      - frame TeachingPoints_16-06-04 at (12133.67, 1957.34, 973.56) mm, rotated rx 180 ry 0 rz 0 deg
        - target Point_16-06-04 (Cartesian target) at (0, 0, 0) mm; joints [12200, 3550, 510] of gantry
      - frame TeachingPoints_17-06-04 at (12633.67, 1957.34, 973.56) mm, rotated rx 180 ry 0 rz 0 deg
        - target Point_17-06-04 (Cartesian target) at (0, 0, 0) mm; joints [12700, 3550, 510] of gantry
      - frame TeachingPoints_18-06-04 at (13133.67, 1957.34, 973.56) mm, rotated rx 180 ry 0 rz 0 deg
        - target Point_18-06-04 (Cartesian target) at (0, 0, 0) mm; joints [13200, 3550, 510] of gantry
      - frame TeachingPoints_19-06-04 at (13633.67, 1957.34, 973.56) mm, rotated rx 180 ry 0 rz 0 deg
        - target Point_19-06-04 (Cartesian target) at (0, 0, 0) mm; joints [13700, 3550, 510] of gantry
      - frame TeachingPoints_20-06-04 at (14133.67, 1957.34, 973.56) mm, rotated rx 180 ry 0 rz 0 deg
        - target Point_20-06-04 (Cartesian target) at (0, 0, 0) mm; joints [14200, 3550, 510] of gantry
      - frame TeachingPoints_01-01-05 at (4633.67, 4457.34, 1108.56) mm, rotated rx 180 ry 0 rz 0 deg
        - target Point_01-01-05 (Cartesian target) at (0, 0, 0) mm; joints [4700, 1050, 375] of gantry
      - frame TeachingPoints_02-01-05 at (5133.67, 4457.34, 1108.56) mm, rotated rx 180 ry 0 rz 0 deg
        - target Point_02-01-05 (Cartesian target) at (0, 0, 0) mm; joints [5200, 1050, 375] of gantry
      - frame TeachingPoints_03-01-05 at (5633.67, 4457.34, 1108.56) mm, rotated rx 180 ry 0 rz 0 deg
        - target Point_03-01-05 (Cartesian target) at (0, 0, 0) mm; joints [5700, 1050, 375] of gantry
      - frame TeachingPoints_04-01-05 at (6133.67, 4457.34, 1108.56) mm, rotated rx 180 ry 0 rz 0 deg
        - target Point_04-01-05 (Cartesian target) at (0, 0, 0) mm; joints [6200, 1050, 375] of gantry
      - frame TeachingPoints_05-01-05 at (6633.67, 4457.34, 1108.56) mm, rotated rx 180 ry 0 rz 0 deg
        - target Point_05-01-05 (Cartesian target) at (0, 0, 0) mm; joints [6700, 1050, 375] of gantry
      - frame TeachingPoints_06-01-05 at (7133.67, 4457.34, 1108.56) mm, rotated rx 180 ry 0 rz 0 deg
        - target Point_06-01-05 (Cartesian target) at (0, 0, 0) mm; joints [7200, 1050, 375] of gantry
      - frame TeachingPoints_07-01-05 at (7633.67, 4457.34, 1108.56) mm, rotated rx 180 ry 0 rz 0 deg
        - target Point_07-01-05 (Cartesian target) at (0, 0, 0) mm; joints [7700, 1050, 375] of gantry
      - frame TeachingPoints_08-01-05 at (8133.67, 4457.34, 1108.56) mm, rotated rx 180 ry 0 rz 0 deg
        - target Point_08-01-05 (Cartesian target) at (0, 0, 0) mm; joints [8200, 1050, 375] of gantry
      - frame TeachingPoints_09-01-05 at (8633.67, 4457.34, 1108.56) mm, rotated rx 180 ry 0 rz 0 deg
        - target Point_09-01-05 (Cartesian target) at (0, 0, 0) mm; joints [8700, 1050, 375] of gantry
      - frame TeachingPoints_10-01-05 at (9133.67, 4457.34, 1108.56) mm, rotated rx 180 ry 0 rz 0 deg
        - target Point_10-01-05 (Cartesian target) at (0, 0, 0) mm; joints [9200, 1050, 375] of gantry
      - frame TeachingPoints_11-01-05 at (9633.67, 4457.34, 1108.56) mm, rotated rx 180 ry 0 rz 0 deg
        - target Point_11-01-05 (Cartesian target) at (0, 0, 0) mm; joints [9700, 1050, 375] of gantry
      - frame TeachingPoints_12-01-05 at (10133.67, 4457.34, 1108.56) mm, rotated rx 180 ry 0 rz 0 deg
        - target Point_12-01-05 (Cartesian target) at (0, 0, 0) mm; joints [10200, 1050, 375] of gantry
      - frame TeachingPoints_13-01-05 at (10633.67, 4457.34, 1108.56) mm, rotated rx 180 ry 0 rz 0 deg
        - target Point_13-01-05 (Cartesian target) at (0, 0, 0) mm; joints [10700, 1050, 375] of gantry
      - frame TeachingPoints_14-01-05 at (11133.67, 4457.34, 1108.56) mm, rotated rx 180 ry 0 rz 0 deg
        - target Point_14-01-05 (Cartesian target) at (0, 0, 0) mm; joints [11200, 1050, 375] of gantry
      - frame TeachingPoints_15-01-05 at (11633.67, 4457.34, 1108.56) mm, rotated rx 180 ry 0 rz 0 deg
        - target Point_15-01-05 (Cartesian target) at (0, 0, 0) mm; joints [11700, 1050, 375] of gantry
      - frame TeachingPoints_16-01-05 at (12133.67, 4457.34, 1108.56) mm, rotated rx 180 ry 0 rz 0 deg
        - target Point_16-01-05 (Cartesian target) at (0, 0, 0) mm; joints [12200, 1050, 375] of gantry
      - frame TeachingPoints_17-01-05 at (12633.67, 4457.34, 1108.56) mm, rotated rx 180 ry 0 rz 0 deg
        - target Point_17-01-05 (Cartesian target) at (0, 0, 0) mm; joints [12700, 1050, 375] of gantry
      - frame TeachingPoints_18-01-05 at (13133.67, 4457.34, 1108.56) mm, rotated rx 180 ry 0 rz 0 deg
        - target Point_18-01-05 (Cartesian target) at (0, 0, 0) mm; joints [13200, 1050, 375] of gantry
      - frame TeachingPoints_19-01-05 at (13633.67, 4457.34, 1108.56) mm, rotated rx 180 ry 0 rz 0 deg
        - target Point_19-01-05 (Cartesian target) at (0, 0, 0) mm; joints [13700, 1050, 375] of gantry
      - frame TeachingPoints_20-01-05 at (14133.67, 4457.34, 1108.56) mm, rotated rx 180 ry 0 rz 0 deg
        - target Point_20-01-05 (Cartesian target) at (0, 0, 0) mm; joints [14200, 1050, 375] of gantry
      - frame TeachingPoints_01-02-05 at (4633.67, 3957.34, 1108.56) mm, rotated rx 180 ry 0 rz 0 deg
        - target Point_01-02-05 (Cartesian target) at (0, 0, 0) mm; joints [4700, 1550, 375] of gantry
      - frame TeachingPoints_02-02-05 at (5133.67, 3957.34, 1108.56) mm, rotated rx 180 ry 0 rz 0 deg
        - target Point_02-02-05 (Cartesian target) at (0, 0, 0) mm; joints [5200, 1550, 375] of gantry
      - frame TeachingPoints_03-02-05 at (5633.67, 3957.34, 1108.56) mm, rotated rx 180 ry 0 rz 0 deg
        - target Point_03-02-05 (Cartesian target) at (0, 0, 0) mm; joints [5700, 1550, 375] of gantry
      - frame TeachingPoints_04-02-05 at (6133.67, 3957.34, 1108.56) mm, rotated rx 180 ry 0 rz 0 deg
        - target Point_04-02-05 (Cartesian target) at (0, 0, 0) mm; joints [6200, 1550, 375] of gantry
      - frame TeachingPoints_05-02-05 at (6633.67, 3957.34, 1108.56) mm, rotated rx 180 ry 0 rz 0 deg
        - target Point_05-02-05 (Cartesian target) at (0, 0, 0) mm; joints [6700, 1550, 375] of gantry
      - frame TeachingPoints_06-02-05 at (7133.67, 3957.34, 1108.56) mm, rotated rx 180 ry 0 rz 0 deg
        - target Point_06-02-05 (Cartesian target) at (0, 0, 0) mm; joints [7200, 1550, 375] of gantry
      - frame TeachingPoints_07-02-05 at (7633.67, 3957.34, 1108.56) mm, rotated rx 180 ry 0 rz 0 deg
        - target Point_07-02-05 (Cartesian target) at (0, 0, 0) mm; joints [7700, 1550, 375] of gantry
      - frame TeachingPoints_08-02-05 at (8133.67, 3957.34, 1108.56) mm, rotated rx 180 ry 0 rz 0 deg
        - target Point_08-02-05 (Cartesian target) at (0, 0, 0) mm; joints [8200, 1550, 375] of gantry
      - frame TeachingPoints_09-02-05 at (8633.67, 3957.34, 1108.56) mm, rotated rx 180 ry 0 rz 0 deg
        - target Point_09-02-05 (Cartesian target) at (0, 0, 0) mm; joints [8700, 1550, 375] of gantry
      - frame TeachingPoints_10-02-05 at (9133.67, 3957.34, 1108.56) mm, rotated rx 180 ry 0 rz 0 deg
        - target Point_10-02-05 (Cartesian target) at (0, 0, 0) mm; joints [9200, 1550, 375] of gantry
      - frame TeachingPoints_11-02-05 at (9633.67, 3957.34, 1108.56) mm, rotated rx 180 ry 0 rz 0 deg
        - target Point_11-02-05 (Cartesian target) at (0, 0, 0) mm; joints [9700, 1550, 375] of gantry
      - frame TeachingPoints_12-02-05 at (10133.67, 3957.34, 1108.56) mm, rotated rx 180 ry 0 rz 0 deg
        - target Point_12-02-05 (Cartesian target) at (0, 0, 0) mm; joints [10200, 1550, 375] of gantry
      - frame TeachingPoints_13-02-05 at (10633.67, 3957.34, 1108.56) mm, rotated rx 180 ry 0 rz 0 deg
        - target Point_13-02-05 (Cartesian target) at (0, 0, 0) mm; joints [10700, 1550, 375] of gantry
      - frame TeachingPoints_14-02-05 at (11133.67, 3957.34, 1108.56) mm, rotated rx 180 ry 0 rz 0 deg
        - target Point_14-02-05 (Cartesian target) at (0, 0, 0) mm; joints [11200, 1550, 375] of gantry
      - frame TeachingPoints_15-02-05 at (11633.67, 3957.34, 1108.56) mm, rotated rx 180 ry 0 rz 0 deg
        - target Point_15-02-05 (Cartesian target) at (0, 0, 0) mm; joints [11700, 1550, 375] of gantry
      - frame TeachingPoints_16-02-05 at (12133.67, 3957.34, 1108.56) mm, rotated rx 180 ry 0 rz 0 deg
        - target Point_16-02-05 (Cartesian target) at (0, 0, 0) mm; joints [12200, 1550, 375] of gantry
      - frame TeachingPoints_17-02-05 at (12633.67, 3957.34, 1108.56) mm, rotated rx 180 ry 0 rz 0 deg
        - target Point_17-02-05 (Cartesian target) at (0, 0, 0) mm; joints [12700, 1550, 375] of gantry
      - frame TeachingPoints_18-02-05 at (13133.67, 3957.34, 1108.56) mm, rotated rx 180 ry 0 rz 0 deg
        - target Point_18-02-05 (Cartesian target) at (0, 0, 0) mm; joints [13200, 1550, 375] of gantry
      - frame TeachingPoints_19-02-05 at (13633.67, 3957.34, 1108.56) mm, rotated rx 180 ry 0 rz 0 deg
        - target Point_19-02-05 (Cartesian target) at (0, 0, 0) mm; joints [13700, 1550, 375] of gantry
      - frame TeachingPoints_20-02-05 at (14133.67, 3957.34, 1108.56) mm, rotated rx 180 ry 0 rz 0 deg
        - target Point_20-02-05 (Cartesian target) at (0, 0, 0) mm; joints [14200, 1550, 375] of gantry
      - frame TeachingPoints_01-03-05 at (4633.67, 3457.34, 1108.56) mm, rotated rx 180 ry 0 rz 0 deg
        - target Point_01-03-05 (Cartesian target) at (0, 0, 0) mm; joints [4700, 2050, 375] of gantry
      - frame TeachingPoints_02-03-05 at (5133.67, 3457.34, 1108.56) mm, rotated rx 180 ry 0 rz 0 deg
        - target Point_02-03-05 (Cartesian target) at (0, 0, 0) mm; joints [5200, 2050, 375] of gantry
      - frame TeachingPoints_03-03-05 at (5633.67, 3457.34, 1108.56) mm, rotated rx 180 ry 0 rz 0 deg
        - target Point_03-03-05 (Cartesian target) at (0, 0, 0) mm; joints [5700, 2050, 375] of gantry
      - frame TeachingPoints_04-03-05 at (6133.67, 3457.34, 1108.56) mm, rotated rx 180 ry 0 rz 0 deg
        - target Point_04-03-05 (Cartesian target) at (0, 0, 0) mm; joints [6200, 2050, 375] of gantry
      - frame TeachingPoints_05-03-05 at (6633.67, 3457.34, 1108.56) mm, rotated rx 180 ry 0 rz 0 deg
        - target Point_05-03-05 (Cartesian target) at (0, 0, 0) mm; joints [6700, 2050, 375] of gantry
      - frame TeachingPoints_06-03-05 at (7133.67, 3457.34, 1108.56) mm, rotated rx 180 ry 0 rz 0 deg
        - target Point_06-03-05 (Cartesian target) at (0, 0, 0) mm; joints [7200, 2050, 375] of gantry
      - frame TeachingPoints_07-03-05 at (7633.67, 3457.34, 1108.56) mm, rotated rx 180 ry 0 rz 0 deg
        - target Point_07-03-05 (Cartesian target) at (0, 0, 0) mm; joints [7700, 2050, 375] of gantry
      - frame TeachingPoints_08-03-05 at (8133.67, 3457.34, 1108.56) mm, rotated rx 180 ry 0 rz 0 deg
        - target Point_08-03-05 (Cartesian target) at (0, 0, 0) mm; joints [8200, 2050, 375] of gantry
      - frame TeachingPoints_09-03-05 at (8633.67, 3457.34, 1108.56) mm, rotated rx 180 ry 0 rz 0 deg
        - target Point_09-03-05 (Cartesian target) at (0, 0, 0) mm; joints [8700, 2050, 375] of gantry
      - frame TeachingPoints_10-03-05 at (9133.67, 3457.34, 1108.56) mm, rotated rx 180 ry 0 rz 0 deg
        - target Point_10-03-05 (Cartesian target) at (0, 0, 0) mm; joints [9200, 2050, 375] of gantry
      - frame TeachingPoints_11-03-05 at (9633.67, 3457.34, 1108.56) mm, rotated rx 180 ry 0 rz 0 deg
        - target Point_11-03-05 (Cartesian target) at (0, 0, 0) mm; joints [9700, 2050, 375] of gantry
      - frame TeachingPoints_12-03-05 at (10133.67, 3457.34, 1108.56) mm, rotated rx 180 ry 0 rz 0 deg
        - target Point_12-03-05 (Cartesian target) at (0, 0, 0) mm; joints [10200, 2050, 375] of gantry
      - frame TeachingPoints_13-03-05 at (10633.67, 3457.34, 1108.56) mm, rotated rx 180 ry 0 rz 0 deg
        - target Point_13-03-05 (Cartesian target) at (0, 0, 0) mm; joints [10700, 2050, 375] of gantry
      - frame TeachingPoints_14-03-05 at (11133.67, 3457.34, 1108.56) mm, rotated rx 180 ry 0 rz 0 deg
        - target Point_14-03-05 (Cartesian target) at (0, 0, 0) mm; joints [11200, 2050, 375] of gantry
      - frame TeachingPoints_15-03-05 at (11633.67, 3457.34, 1108.56) mm, rotated rx 180 ry 0 rz 0 deg
        - target Point_15-03-05 (Cartesian target) at (0, 0, 0) mm; joints [11700, 2050, 375] of gantry
      - frame TeachingPoints_16-03-05 at (12133.67, 3457.34, 1108.56) mm, rotated rx 180 ry 0 rz 0 deg
        - target Point_16-03-05 (Cartesian target) at (0, 0, 0) mm; joints [12200, 2050, 375] of gantry
      - frame TeachingPoints_17-03-05 at (12633.67, 3457.34, 1108.56) mm, rotated rx 180 ry 0 rz 0 deg
        - target Point_17-03-05 (Cartesian target) at (0, 0, 0) mm; joints [12700, 2050, 375] of gantry
      - frame TeachingPoints_18-03-05 at (13133.67, 3457.34, 1108.56) mm, rotated rx 180 ry 0 rz 0 deg
        - target Point_18-03-05 (Cartesian target) at (0, 0, 0) mm; joints [13200, 2050, 375] of gantry
      - frame TeachingPoints_19-03-05 at (13633.67, 3457.34, 1108.56) mm, rotated rx 180 ry 0 rz 0 deg
        - target Point_19-03-05 (Cartesian target) at (0, 0, 0) mm; joints [13700, 2050, 375] of gantry
      - frame TeachingPoints_20-03-05 at (14133.67, 3457.34, 1108.56) mm, rotated rx 180 ry 0 rz 0 deg
        - target Point_20-03-05 (Cartesian target) at (0, 0, 0) mm; joints [14200, 2050, 375] of gantry
      - frame TeachingPoints_01-04-05 at (4633.67, 2957.34, 1108.56) mm, rotated rx 180 ry 0 rz 0 deg
        - target Point_01-04-05 (Cartesian target) at (0, 0, 0) mm; joints [4700, 2550, 375] of gantry
      - frame TeachingPoints_02-04-05 at (5133.67, 2957.34, 1108.56) mm, rotated rx 180 ry 0 rz 0 deg
        - target Point_02-04-05 (Cartesian target) at (0, 0, 0) mm; joints [5200, 2550, 375] of gantry
      - frame TeachingPoints_03-04-05 at (5633.67, 2957.34, 1108.56) mm, rotated rx 180 ry 0 rz 0 deg
        - target Point_03-04-05 (Cartesian target) at (0, 0, 0) mm; joints [5700, 2550, 375] of gantry
      - frame TeachingPoints_04-04-05 at (6133.67, 2957.34, 1108.56) mm, rotated rx 180 ry 0 rz 0 deg
        - target Point_04-04-05 (Cartesian target) at (0, 0, 0) mm; joints [6200, 2550, 375] of gantry
      - frame TeachingPoints_05-04-05 at (6633.67, 2957.34, 1108.56) mm, rotated rx 180 ry 0 rz 0 deg
        - target Point_05-04-05 (Cartesian target) at (0, 0, 0) mm; joints [6700, 2550, 375] of gantry
      - frame TeachingPoints_06-04-05 at (7133.67, 2957.34, 1108.56) mm, rotated rx 180 ry 0 rz 0 deg
        - target Point_06-04-05 (Cartesian target) at (0, 0, 0) mm; joints [7200, 2550, 375] of gantry
      - frame TeachingPoints_07-04-05 at (7633.67, 2957.34, 1108.56) mm, rotated rx 180 ry 0 rz 0 deg
        - target Point_07-04-05 (Cartesian target) at (0, 0, 0) mm; joints [7700, 2550, 375] of gantry
      - frame TeachingPoints_08-04-05 at (8133.67, 2957.34, 1108.56) mm, rotated rx 180 ry 0 rz 0 deg
        - target Point_08-04-05 (Cartesian target) at (0, 0, 0) mm; joints [8200, 2550, 375] of gantry
      - frame TeachingPoints_09-04-05 at (8633.67, 2957.34, 1108.56) mm, rotated rx 180 ry 0 rz 0 deg
        - target Point_09-04-05 (Cartesian target) at (0, 0, 0) mm; joints [8700, 2550, 375] of gantry
      - frame TeachingPoints_10-04-05 at (9133.67, 2957.34, 1108.56) mm, rotated rx 180 ry 0 rz 0 deg
        - target Point_10-04-05 (Cartesian target) at (0, 0, 0) mm; joints [9200, 2550, 375] of gantry
      - frame TeachingPoints_11-04-05 at (9633.67, 2957.34, 1108.56) mm, rotated rx 180 ry 0 rz 0 deg
        - target Point_11-04-05 (Cartesian target) at (0, 0, 0) mm; joints [9700, 2550, 375] of gantry
      - frame TeachingPoints_12-04-05 at (10133.67, 2957.34, 1108.56) mm, rotated rx 180 ry 0 rz 0 deg
        - target Point_12-04-05 (Cartesian target) at (0, 0, 0) mm; joints [10200, 2550, 375] of gantry
      - frame TeachingPoints_13-04-05 at (10633.67, 2957.34, 1108.56) mm, rotated rx 180 ry 0 rz 0 deg
        - target Point_13-04-05 (Cartesian target) at (0, 0, 0) mm; joints [10700, 2550, 375] of gantry
      - frame TeachingPoints_14-04-05 at (11133.67, 2957.34, 1108.56) mm, rotated rx 180 ry 0 rz 0 deg
        - target Point_14-04-05 (Cartesian target) at (0, 0, 0) mm; joints [11200, 2550, 375] of gantry
      - frame TeachingPoints_15-04-05 at (11633.67, 2957.34, 1108.56) mm, rotated rx 180 ry 0 rz 0 deg
        - target Point_15-04-05 (Cartesian target) at (0, 0, 0) mm; joints [11700, 2550, 375] of gantry
      - frame TeachingPoints_16-04-05 at (12133.67, 2957.34, 1108.56) mm, rotated rx 180 ry 0 rz 0 deg
        - target Point_16-04-05 (Cartesian target) at (0, 0, 0) mm; joints [12200, 2550, 375] of gantry
      - frame TeachingPoints_17-04-05 at (12633.67, 2957.34, 1108.56) mm, rotated rx 180 ry 0 rz 0 deg
        - target Point_17-04-05 (Cartesian target) at (0, 0, 0) mm; joints [12700, 2550, 375] of gantry
      - frame TeachingPoints_18-04-05 at (13133.67, 2957.34, 1108.56) mm, rotated rx 180 ry 0 rz 0 deg
        - target Point_18-04-05 (Cartesian target) at (0, 0, 0) mm; joints [13200, 2550, 375] of gantry
      - frame TeachingPoints_19-04-05 at (13633.67, 2957.34, 1108.56) mm, rotated rx 180 ry 0 rz 0 deg
        - target Point_19-04-05 (Cartesian target) at (0, 0, 0) mm; joints [13700, 2550, 375] of gantry
      - frame TeachingPoints_20-04-05 at (14133.67, 2957.34, 1108.56) mm, rotated rx 180 ry 0 rz 0 deg
        - target Point_20-04-05 (Cartesian target) at (0, 0, 0) mm; joints [14200, 2550, 375] of gantry
      - frame TeachingPoints_01-05-05 at (4633.67, 2457.34, 1108.56) mm, rotated rx 180 ry 0 rz 0 deg
        - target Point_01-05-05 (Cartesian target) at (0, 0, 0) mm; joints [4700, 3050, 375] of gantry
      - frame TeachingPoints_02-05-05 at (5133.67, 2457.34, 1108.56) mm, rotated rx 180 ry 0 rz 0 deg
        - target Point_02-05-05 (Cartesian target) at (0, 0, 0) mm; joints [5200, 3050, 375] of gantry
      - frame TeachingPoints_03-05-05 at (5633.67, 2457.34, 1108.56) mm, rotated rx 180 ry 0 rz 0 deg
        - target Point_03-05-05 (Cartesian target) at (0, 0, 0) mm; joints [5700, 3050, 375] of gantry
      - frame TeachingPoints_04-05-05 at (6133.67, 2457.34, 1108.56) mm, rotated rx 180 ry 0 rz 0 deg
        - target Point_04-05-05 (Cartesian target) at (0, 0, 0) mm; joints [6200, 3050, 375] of gantry
      - frame TeachingPoints_05-05-05 at (6633.67, 2457.34, 1108.56) mm, rotated rx 180 ry 0 rz 0 deg
        - target Point_05-05-05 (Cartesian target) at (0, 0, 0) mm; joints [6700, 3050, 375] of gantry
      - frame TeachingPoints_06-05-05 at (7133.67, 2457.34, 1108.56) mm, rotated rx 180 ry 0 rz 0 deg
        - target Point_06-05-05 (Cartesian target) at (0, 0, 0) mm; joints [7200, 3050, 375] of gantry
      - frame TeachingPoints_07-05-05 at (7633.67, 2457.34, 1108.56) mm, rotated rx 180 ry 0 rz 0 deg
        - target Point_07-05-05 (Cartesian target) at (0, 0, 0) mm; joints [7700, 3050, 375] of gantry
      - frame TeachingPoints_08-05-05 at (8133.67, 2457.34, 1108.56) mm, rotated rx 180 ry 0 rz 0 deg
        - target Point_08-05-05 (Cartesian target) at (0, 0, 0) mm; joints [8200, 3050, 375] of gantry
      - frame TeachingPoints_09-05-05 at (8633.67, 2457.34, 1108.56) mm, rotated rx 180 ry 0 rz 0 deg
        - target Point_09-05-05 (Cartesian target) at (0, 0, 0) mm; joints [8700, 3050, 375] of gantry
      - frame TeachingPoints_10-05-05 at (9133.67, 2457.34, 1108.56) mm, rotated rx 180 ry 0 rz 0 deg
        - target Point_10-05-05 (Cartesian target) at (0, 0, 0) mm; joints [9200, 3050, 375] of gantry
      - frame TeachingPoints_11-05-05 at (9633.67, 2457.34, 1108.56) mm, rotated rx 180 ry 0 rz 0 deg
        - target Point_11-05-05 (Cartesian target) at (0, 0, 0) mm; joints [9700, 3050, 375] of gantry
      - frame TeachingPoints_12-05-05 at (10133.67, 2457.34, 1108.56) mm, rotated rx 180 ry 0 rz 0 deg
        - target Point_12-05-05 (Cartesian target) at (0, 0, 0) mm; joints [10200, 3050, 375] of gantry
      - frame TeachingPoints_13-05-05 at (10633.67, 2457.34, 1108.56) mm, rotated rx 180 ry 0 rz 0 deg
        - target Point_13-05-05 (Cartesian target) at (0, 0, 0) mm; joints [10700, 3050, 375] of gantry
      - frame TeachingPoints_14-05-05 at (11133.67, 2457.34, 1108.56) mm, rotated rx 180 ry 0 rz 0 deg
        - target Point_14-05-05 (Cartesian target) at (0, 0, 0) mm; joints [11200, 3050, 375] of gantry
      - frame TeachingPoints_15-05-05 at (11633.67, 2457.34, 1108.56) mm, rotated rx 180 ry 0 rz 0 deg
        - target Point_15-05-05 (Cartesian target) at (0, 0, 0) mm; joints [11700, 3050, 375] of gantry
      - frame TeachingPoints_16-05-05 at (12133.67, 2457.34, 1108.56) mm, rotated rx 180 ry 0 rz 0 deg
        - target Point_16-05-05 (Cartesian target) at (0, 0, 0) mm; joints [12200, 3050, 375] of gantry
      - frame TeachingPoints_17-05-05 at (12633.67, 2457.34, 1108.56) mm, rotated rx 180 ry 0 rz 0 deg
        - target Point_17-05-05 (Cartesian target) at (0, 0, 0) mm; joints [12700, 3050, 375] of gantry
      - frame TeachingPoints_18-05-05 at (13133.67, 2457.34, 1108.56) mm, rotated rx 180 ry 0 rz 0 deg
        - target Point_18-05-05 (Cartesian target) at (0, 0, 0) mm; joints [13200, 3050, 375] of gantry
      - frame TeachingPoints_19-05-05 at (13633.67, 2457.34, 1108.56) mm, rotated rx 180 ry 0 rz 0 deg
        - target Point_19-05-05 (Cartesian target) at (0, 0, 0) mm; joints [13700, 3050, 375] of gantry
      - frame TeachingPoints_20-05-05 at (14133.67, 2457.34, 1108.56) mm, rotated rx 180 ry 0 rz 0 deg
        - target Point_20-05-05 (Cartesian target) at (0, 0, 0) mm; joints [14200, 3050, 375] of gantry
      - frame TeachingPoints_01-06-05 at (4633.67, 1957.34, 1108.56) mm, rotated rx 180 ry 0 rz 0 deg
        - target Point_01-06-05 (Cartesian target) at (0, 0, 0) mm; joints [4700, 3550, 375] of gantry
      - frame TeachingPoints_02-06-05 at (5133.67, 1957.34, 1108.56) mm, rotated rx 180 ry 0 rz 0 deg
        - target Point_02-06-05 (Cartesian target) at (0, 0, 0) mm; joints [5200, 3550, 375] of gantry
      - frame TeachingPoints_03-06-05 at (5633.67, 1957.34, 1108.56) mm, rotated rx 180 ry 0 rz 0 deg
        - target Point_03-06-05 (Cartesian target) at (0, 0, 0) mm; joints [5700, 3550, 375] of gantry
      - frame TeachingPoints_04-06-05 at (6133.67, 1957.34, 1108.56) mm, rotated rx 180 ry 0 rz 0 deg
        - target Point_04-06-05 (Cartesian target) at (0, 0, 0) mm; joints [6200, 3550, 375] of gantry
      - frame TeachingPoints_05-06-05 at (6633.67, 1957.34, 1108.56) mm, rotated rx 180 ry 0 rz 0 deg
        - target Point_05-06-05 (Cartesian target) at (0, 0, 0) mm; joints [6700, 3550, 375] of gantry
      - frame TeachingPoints_06-06-05 at (7133.67, 1957.34, 1108.56) mm, rotated rx 180 ry 0 rz 0 deg
        - target Point_06-06-05 (Cartesian target) at (0, 0, 0) mm; joints [7200, 3550, 375] of gantry
      - frame TeachingPoints_07-06-05 at (7633.67, 1957.34, 1108.56) mm, rotated rx 180 ry 0 rz 0 deg
        - target Point_07-06-05 (Cartesian target) at (0, 0, 0) mm; joints [7700, 3550, 375] of gantry
      - frame TeachingPoints_08-06-05 at (8133.67, 1957.34, 1108.56) mm, rotated rx 180 ry 0 rz 0 deg
        - target Point_08-06-05 (Cartesian target) at (0, 0, 0) mm; joints [8200, 3550, 375] of gantry
      - frame TeachingPoints_09-06-05 at (8633.67, 1957.34, 1108.56) mm, rotated rx 180 ry 0 rz 0 deg
        - target Point_09-06-05 (Cartesian target) at (0, 0, 0) mm; joints [8700, 3550, 375] of gantry
      - frame TeachingPoints_10-06-05 at (9133.67, 1957.34, 1108.56) mm, rotated rx 180 ry 0 rz 0 deg
        - target Point_10-06-05 (Cartesian target) at (0, 0, 0) mm; joints [9200, 3550, 375] of gantry
      - frame TeachingPoints_11-06-05 at (9633.67, 1957.34, 1108.56) mm, rotated rx 180 ry 0 rz 0 deg
        - target Point_11-06-05 (Cartesian target) at (0, 0, 0) mm; joints [9700, 3550, 375] of gantry
      - frame TeachingPoints_12-06-05 at (10133.67, 1957.34, 1108.56) mm, rotated rx 180 ry 0 rz 0 deg
        - target Point_12-06-05 (Cartesian target) at (0, 0, 0) mm; joints [10200, 3550, 375] of gantry
      - frame TeachingPoints_13-06-05 at (10633.67, 1957.34, 1108.56) mm, rotated rx 180 ry 0 rz 0 deg
        - target Point_13-06-05 (Cartesian target) at (0, 0, 0) mm; joints [10700, 3550, 375] of gantry
      - frame TeachingPoints_14-06-05 at (11133.67, 1957.34, 1108.56) mm, rotated rx 180 ry 0 rz 0 deg
        - target Point_14-06-05 (Cartesian target) at (0, 0, 0) mm; joints [11200, 3550, 375] of gantry
      - frame TeachingPoints_15-06-05 at (11633.67, 1957.34, 1108.56) mm, rotated rx 180 ry 0 rz 0 deg
        - target Point_15-06-05 (Cartesian target) at (0, 0, 0) mm; joints [11700, 3550, 375] of gantry
      - frame TeachingPoints_16-06-05 at (12133.67, 1957.34, 1108.56) mm, rotated rx 180 ry 0 rz 0 deg
        - target Point_16-06-05 (Cartesian target) at (0, 0, 0) mm; joints [12200, 3550, 375] of gantry
      - frame TeachingPoints_17-06-05 at (12633.67, 1957.34, 1108.56) mm, rotated rx 180 ry 0 rz 0 deg
        - target Point_17-06-05 (Cartesian target) at (0, 0, 0) mm; joints [12700, 3550, 375] of gantry
      - frame TeachingPoints_18-06-05 at (13133.67, 1957.34, 1108.56) mm, rotated rx 180 ry 0 rz 0 deg
        - target Point_18-06-05 (Cartesian target) at (0, 0, 0) mm; joints [13200, 3550, 375] of gantry
      - frame TeachingPoints_19-06-05 at (13633.67, 1957.34, 1108.56) mm, rotated rx 180 ry 0 rz 0 deg
        - target Point_19-06-05 (Cartesian target) at (0, 0, 0) mm; joints [13700, 3550, 375] of gantry
      - frame TeachingPoints_20-06-05 at (14133.67, 1957.34, 1108.56) mm, rotated rx 180 ry 0 rz 0 deg
        - target Point_20-06-05 (Cartesian target) at (0, 0, 0) mm; joints [14200, 3550, 375] of gantry
  - frame Frame 36 at (12000, 3370, 2800) mm, rotated rx -105 ry 0 rz 90 deg
  - camera Camera 1
